FUNCTION_BLOCK Modulate
VAR
	_CurrentImage : ITcVnImage;
	_unwrapper	  : I_Unwrapper;
	value		  : HRESULT;
END_VAR

PROPERTY PUBLIC CurrentFrameImage : ITcVnImage
GET
CurrentFrameImage := _CurrentImage;
END_GET
END_PROPERTY

//FB_Init is always available implicitly and it is used primarily for initialization.
//The return value is not evaluated. For a specific influence, you can also declare the
//methods explicitly and provide additional code there with the standard initialization
//code. You can evaluate the return value.
METHOD FB_Init: BOOL
VAR_INPUT
    bInitRetains: BOOL; // TRUE: the retain variables are initialized (reset warm / reset cold)
    bInCopyCode: BOOL;  // TRUE: the instance will be copied to the copy code afterward (online change)
    Width: UDINT;       // Output image buffer width — pass GVL.STRIP_LENGTH
END_VAR
F_VN_CreateImage(_CurrentImage,
				 Width,
				 1,
				 ETcVnElementType.TCVN_ET_USINT,
				 4,
				 S_OK);
END_METHOD

METHOD GetImage
VAR_INPUT
	Source					  : ITcVnImage;
	SourceWidth, SourceHeight : UDINT;
	OutputWidth, OutputHeight : UDINT;
	OffsetX, Offsety		  : UDINT;
END_VAR

VAR
	x, y			   : UDINT;
	_SampleX, _SampleY : UDINT;
	currentPixel	   : TcVnVector4_LREAL;
END_VAR
FOR y := 0 TO OutputHeight - 1 DO
	FOR x := 0 TO OutputWidth - 1 DO
		_unwrapper.Sample(ImageWidth  := SourceWidth,
						  ImageHeight := SourceHeight,
						  XOffset	  := x + OffsetX,
						  YOffset	  := y + OffsetY);

		IF SUCCEEDED(F_VN_GetPixel(ipSrcImage := Source,
								   aValue	  := currentPixel,
								   nX		  := _unwrapper.X,
								   nY		  := _unwrapper.Y,
								   hrPrev	  := s_OK)) THEN
			value := F_VN_SetPixel(ipSrcImage := _CurrentImage,
						  aValue	 := currentPixel,
						  nX		 := x,
						  nY		 := y,
						  hrPrev	 := s_OK);
		END_IF
	END_FOR
END_FOR
END_METHOD

PROPERTY Unwrapper : I_Unwrapper
GET
Unwrapper := _unwrapper;
END_GET
SET
_unwrapper := Unwrapper;
END_SET
END_PROPERTY

END_FUNCTION_BLOCK

(* stored: Version 1.1.0.1
   POU Modulate: Id {5350d40a-0c99-4bbb-83b2-ad11dbf9cb22}, SpecialFunc None
   Property CurrentFrameImage: Id {eea89cec-a60c-4fd9-a76b-4f0decd5b30b}
   Get Get: Id {0204719f-9ecb-4743-89f7-7cfaee20f1de}
   Method FB_Init: Id {46693cb2-f04a-4e2d-b7c3-ec23a9b28894}
   Method GetImage: Id {cd891bbb-ad5b-4475-91e7-4fc7008d9e4f}
   Property Unwrapper: Id {5bce6a1b-e709-4e68-b638-d83ded7800df}
   Get Get: Id {69113d6b-e58a-473b-9cbb-19dfb376c683}
   Set Set: Id {e11ff1bf-5847-4617-ba21-617cec436575} *)
